// TIA Portal V20 export
FUNCTION "ModuleDiag" : Void   // FC82, SCL
{ S7_Optimized_Access := 'TRUE' }
VERSION : 1.1
// stored: SetENOAutomatically false
   VAR_INPUT
      errorCode : Word;   // Code of error
      value : Bool;   // TRUE for incoming / FALSE for outgoing
   END_VAR
   VAR_IN_OUT
      diag : "typeModuleDiag";   // Diagnostics by module
      errorCounter : USInt;   // Error counter (different errors only)
   END_VAR
BEGIN
   //=============================================================================
   // SIEMENS AG
   // (c)Copyright 2017
   //-----------------------------------------------------------------------------
   // Library:       -
   // Tested with:   CPU 1211C FW V4.2 and ET200SP (IM 155-6 PN BA + AQ 4xU/I ST)
   // Engineering:   TIA Portal V14 Update1
   // Restrictions:  call in FB "1x00Diag82"
   // Requirements:  SIMATIC S7-1200 or S7-1500 CPU
   // Functionality: Module diagnostics (PROFINET IO or central I/O)
   //-----------------------------------------------------------------------------
   // Change log table:
   // Version  Date        Expert in charge                 Changes applied
   // 02.00.00 12.01.2016  SIMATIC Industry Online Support  New function: ModuleDiag
   //=============================================================================

   CASE WORD_TO_INT(#errorCode) OF // errorCode identifier
     1:
       #diag.shortCircuit := #value;

     6:
       #diag.wireBreak := #value;

     7:
       #diag.highLimitExceeded := #value;

     8:
       #diag.lowLimitExceeded := #value;

     17:
       #diag.noSupplyVoltage := #value;
   END_CASE;

   IF (#value = TRUE) THEN // errorCounter (different errors only)
     #errorCounter := #errorCounter + 1;
   ELSE
     #errorCounter := #errorCounter - 1;
   END_IF;
END_FUNCTION
